// SIMATIC S7-200 project (STEP 7-Micro/WIN), CPU 224XP REL 02.01

SYMBOL_TABLE USER2
RED_1            Q0.0
YEL_1            Q0.1
GRE_1            Q0.2
RED_2            Q0.5
YEL_2            Q0.6
GRE_2            Q0.7
Delay_1          VW10
Delay_2          VW12
END_SYMBOL_TABLE

SYMBOL_TABLE S7-200 Symbols
Always_On        SM0.0    // Always ON
First_Scan_On    SM0.1    // ON for the first scan cycle only
Pot0_Value       SMB28    // Set to value corresponding to analog adjustment 0.
Pot1_Value       SMB29    // Set to value corresponding to analog adjustment 1.
END_SYMBOL_TABLE

ORGANIZATION_BLOCK MAIN:OB1
TITLE=PROGRAM COMMENTS
BEGIN
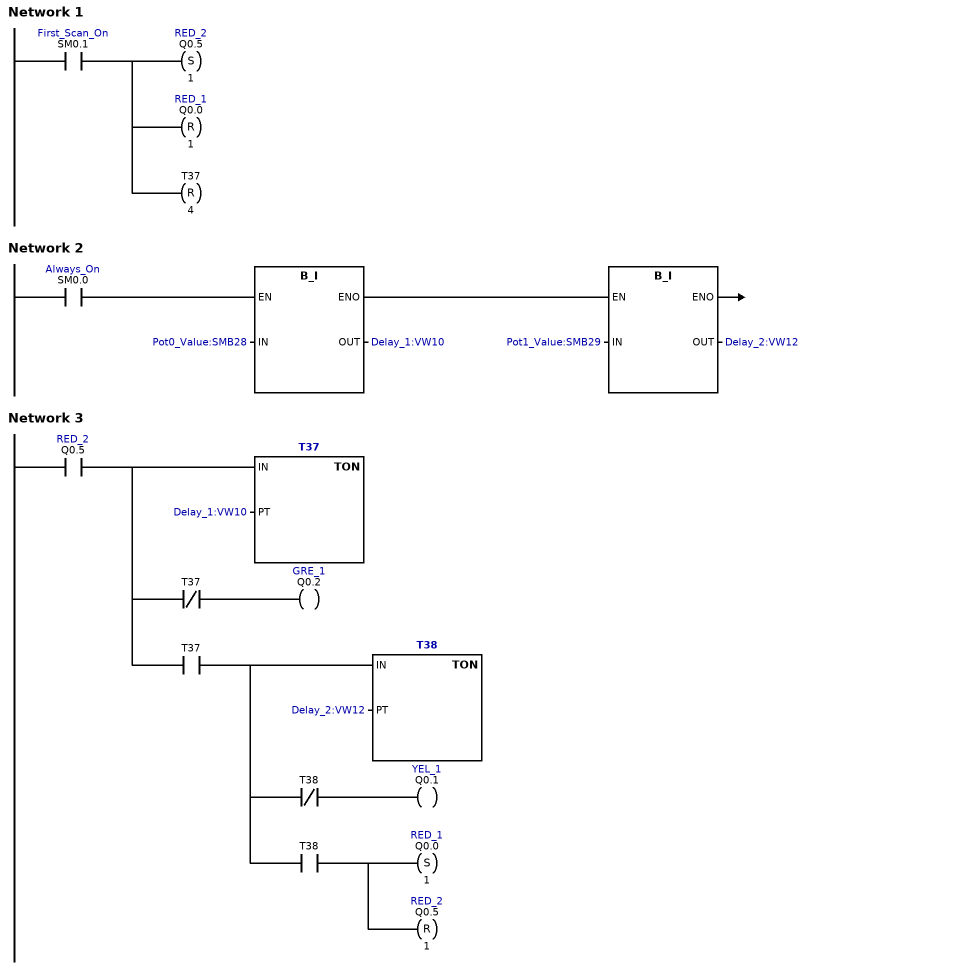
Network 1
LD     First_Scan_On:SM0.1
S      RED_2:Q0.5, 1
R      RED_1:Q0.0, 1
R      T37, 4
Network 2
LD     Always_On:SM0.0
BTI    Pot0_Value:SMB28, Delay_1:VW10
AENO
BTI    Pot1_Value:SMB29, Delay_2:VW12
Network 3
// (network saved uncompiled; LAD cells follow)
// row 0: c0 -| |- RED_2:Q0.5 v  c1 --  c2 [TON T37 IN:=power@row0, PT:=Delay_1:VW10]
// row 1: c0 ^v  c2 [box]
// row 2: c0 ^v  c1 -|/|- T37  c2 -( ) GRE_1:Q0.2
// row 3: c0 ^  c1 -| |- T37 v  c2 --  c3 [TON T38 IN:=power@row3, PT:=Delay_2:VW12]
// row 4: c1 ^v  c3 [box]
// row 5: c1 ^v  c2 -|/|- T38  c3 -( ) YEL_1:Q0.1
// row 6: c1 ^  c2 -| |- T38 v  c3 -(S) RED_1:Q0.0, 1
// row 7: c2 ^  c3 -(R) RED_2:Q0.5, 1
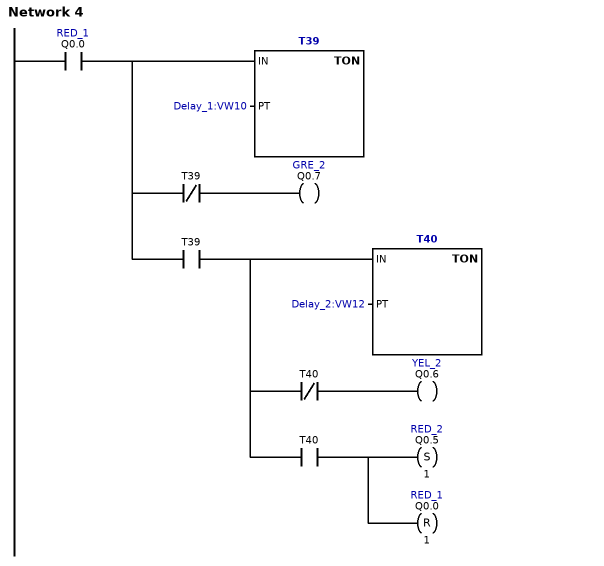
Network 4
// (network saved uncompiled; LAD cells follow)
// row 0: c0 -| |- RED_1:Q0.0 v  c1 --  c2 [TON T39 IN:=power@row0, PT:=Delay_1:VW10]
// row 1: c0 ^v  c2 [box]
// row 2: c0 ^v  c1 -|/|- T39  c2 -( ) GRE_2:Q0.7
// row 3: c0 ^  c1 -| |- T39 v  c2 --  c3 [TON T40 IN:=power@row3, PT:=Delay_2:VW12]
// row 4: c1 ^v  c3 [box]
// row 5: c1 ^v  c2 -|/|- T40  c3 -( ) YEL_2:Q0.6
// row 6: c1 ^  c2 -| |- T40 v  c3 -(S) RED_2:Q0.5, 1
// row 7: c2 ^  c3 -(R) RED_1:Q0.0, 1
END_ORGANIZATION_BLOCK
